// TwinCAT 3 PLC project PLC3
// ProgramVersion: 3.1.4022.3
// libraries:
//   Tc2_Standard, * (Beckhoff Automation GmbH)
//   Tc2_System, * (Beckhoff Automation GmbH)
//   Tc3_Module, * (Beckhoff Automation GmbH)
// project tree:
//   / CheckStatus.TcPOU, GlobalTextList.TcGTLO (not stored), PlcTask.TcTTO (not stored), Visualization Manager.TcVMO (not stored)
//   DUTs/ States.TcDUT
//   GVLs/ GVL_IO.TcGVL (not stored)
//   POUs/ MAIN.TcPOU, MoveArm.TcPOU

// ---- DUTs/States.TcDUT
{attribute 'qualified_only'}
{attribute 'strict'}
TYPE States :
(
	Init := 0,
	Idle,
	MoveToPickUp,
	PickUpDown,
	PickUpUp,
	Moving,
	DropDown,
	DropUp,
	PalletFull
);
END_TYPE

// ---- CheckStatus.TcPOU
FUNCTION_BLOCK CheckStatus
VAR_INPUT
	Position :INT;
	InputArray: ARRAY [1..25] OF BOOL;
END_VAR
VAR_OUTPUT
Occupied : BOOL;
END_VAR

Occupied := FALSE;
IF InputArray[Position] THEN
	Occupied := TRUE;
END_IF

END_FUNCTION_BLOCK

// ---- POUs/MAIN.TcPOU
PROGRAM MAIN
VAR
	Timer1 :TON;
	Timer2 : TON;
	Timer3 : TON;
	PulseTimer1 : TP;

	CurrentState  : States;
	
	ServoRTrigY : R_Trig ; 
	ServoRTrigX : R_Trig ; 
	
	//Eigen trigger booleans
	InitYReady : BOOL;
	InitXReady : BOOL;
	droppingDown : BOOL; //test
	
	TimerTest1 : TIME;
	TimerResult : TIME;
	
	Move_Arm : MoveArm;
	Check_Status : CheckStatus;
	
	PalletArray: ARRAY [1..25] OF BOOL := [25(FALSE)];

	Pos : INT;
END_VAR

PulseTimer1(IN:=GVL_IO.Start_button, PT:=T#150MS);
Timer1(IN:= GVL_IO.a_1_Vertical_Zaxis_downward, PT:= T#10MS);
Timer2(IN:=GVL_IO.a_1_Vertical_Zaxis_downward, PT:=T#10MS);
Timer3(IN:=droppingDown AND NOT GVL_IO.a_1_Vertical_Zaxis_downward, PT:=T#280MS);

CASE CurrentState OF
States.Init:
		//Aanzetten van servo's. Dit kan even duren GEEN HOMING
		GVL_IO.SVONX_SERVO_ON_tableX 	  := TRUE; 
		GVL_IO.SVONY_SERVO_ON_translY 	  := TRUE;
		
		GVL_IO.SETUPX_ORIGIN_tableX := PulseTimer1.Q;
		GVL_IO.SETUPY_ORIGIN_translY := PulseTimer1.Q;
		
		//// Koppelen van outputs Busy aan var's. Triggered op een falling edge.
		IF PulseTimer1.Q THEN
			ServoRTrigX ( clk := gvl_io.SETONX_ORIGIN_tableX ); 
	  		ServoRTrigY ( clk := gvl_io.SETONY_ORIGIN_translationY );
		END_IF
		
		// Bools setten aan de hand van triggers.
		IF ServoRTrigX.Q THEN
			InitXReady:= TRUE;
		END_IF
		
		IF ServoRTrigY.Q THEN
			InitYReady:= TRUE;
		END_IF
		
		// Init voltooid ga naar idle
		IF InitXReady AND InitYReady THEN
			Pos:= 1;
			CurrentState:= States.Idle;
		END_IF
		
States.Idle:
		IF NOT GVL_IO.Stop_button AND NOT GVL_IO.dp2_Cover_detection THEN
			//SEND MESSAGEE TODO
			CurrentState := States.Idle;
		END_IF
		
		IF NOT GVL_IO.Stop_button AND GVL_IO.dp1_Can_detection AND GVL_IO.dp2_Cover_detection THEN
			CurrentState := States.MoveToPickUp;
		END_IF
		
States.MoveToPickUp:
		Check_Status(Position:= POS, InputArray:= PalletArray);
		IF Check_Status.Occupied THEN
			CurrentState := States.ManualCheck;
			ELSE
				Move_Arm(Position:= 30);
				IF Move_Arm.OnNewLocation THEN
				CurrentState := States.PickUpDown;
				END_IF
		END_IF
		
States.PickUpDown:
		IF GVL_IO.a_0_Vertical_Zaxis_upward THEN
			GVL_IO.Aplus_Vert_axis_downwards := TRUE;
		END_IF
		
		IF GVL_IO.a_1_Vertical_Zaxis_downward THEN
			GVL_IO.Vplus_Vacuum_start := TRUE;
			
			IF Timer1.Q THEN
			CurrentState := States.PickUpUp;
			END_IF
		END_IF

States.PickUpUp:
		GVL_IO.Aplus_Vert_axis_downwards := FALSE;
		
		IF GVL_IO.a_0_Vertical_Zaxis_upward THEN
			CurrentState := States.Moving;
		END_IF
		
States.Moving:
		IF GVL_IO.a_0_Vertical_Zaxis_upward THEN
		
		Move_Arm(Position:= Pos);
		IF Move_Arm.OnNewLocation THEN
			PalletArray[Pos] := TRUE; // TEMP Cihan
			CurrentState := States.DropDown;
		END_IF
		END_IF
		
States.DropDown:
		IF GVL_IO.a_0_Vertical_Zaxis_upward THEN
			GVL_IO.Aplus_Vert_axis_downwards := TRUE;
			droppingDown := TRUE;
			TimerTest1 := TIME();
		END_IF
		
		
		IF 	GVL_IO.a_1_Vertical_Zaxis_downward THEN
			GVL_IO.Vplus_Vacuum_start := FALSE;
			IF Timer2.Q THEN
				TimerResult := TIME() - TimerTest1;
				droppingDown := FALSE;
				CurrentState := States.DropUp;
			END_IF
			
		ELSE IF Timer3.Q  THEN
		GVL_io.Aplus_Vert_axis_downwards := FALSE;
		droppingDown := FALSE;
		CurrentState := States.ManualCheck;
		END_IF
		END_IF

States.DropUp:
		IF GVL_IO.a_1_Vertical_Zaxis_downward THEN
			GVL_IO.Aplus_Vert_axis_downwards := FALSE;
		END_IF
		
		IF GVL_IO.a_0_Vertical_Zaxis_upward THEN
			CurrentState := States.Idle;
		END_IF
		
States.ManualCheck:
		GVL_IO.BR_Alarm_light := TRUE;
		GVL_io.Vplus_Vacuum_start := FALSE;
		IF GVL_IO.Reset_button THEN
			GVL_IO.BR_Alarm_light := FALSE;
			Currentstate := States.Idle;
		END_IF
END_CASE

END_PROGRAM

// ---- POUs/MoveArm.TcPOU
FUNCTION_BLOCK MoveArm
VAR_INPUT
Position: INT;
END_VAR
VAR_OUTPUT
	OnNewLocation:BOOL;
END_VAR
VAR
	X: INT;
	Y: INT;
	StartTimer:BOOL;
	
	
	PulseTimer2: TP;
	BusyFtrigX : F_Trig;
	BusyFtrigY : F_Trig;
	ReadyX : BOOL;
	ReadyY : BOOL;
	Busy: BOOL;
END_VAR

OnNewLocation := FALSE;

IF( Position < 1 OR Position > 30)  
	THEN RETURN; 
END_IF

// Calculate X & Y position on Palletiser
// 
X := (Position - 1) MOD 5;

// Position-1 / 5 with ROUND to floor 
Y := ((Position -1) / 5) - ((Position -1) / 5) MOD 1;

// set position 
GVL_IO.INX0_from_Input0_tableX:= X.0;
GVL_IO.INX1_from_Input1_tableX:= X.1;
GVL_IO.INX2_from_Input2_tableX:= X.2;
GVL_IO.INY0_from_Input0_translY:= Y.0;
GVL_IO.INY1_from_Input1_translY:= Y.1;
GVL_IO.INY2_from_Input2_translY:= Y.2;



PulseTimer2(IN:=StartTimer, PT:=T#150MS);

GVL_IO.DRIVEX_MOVE_tableX := PulseTimer2.Q;
GVL_IO.DRIVEY_MOVE_translY := PulseTimer2.Q;
StartTimer:= TRUE;
		
BusyFtrigX ( clk := gvl_io.BUSYX_BUSY_tableX ); 
BusyFtrigY ( clk := gvl_io.BUSYY_BUSY_traslationY );
		
IF BusyFtrigX.Q THEN
	ReadyX:= TRUE;
END_IF
		
IF BusyFtrigY.Q THEN
	ReadyY:= TRUE;
END_IF
		
IF ReadyY AND ReadyX THEN
	GVL_IO.DRIVEX_MOVE_tableX := FALSE;
	GVL_IO.DRIVEY_MOVE_translY := FALSE;
	ReadyX:= FALSE;
	ReadyY:= FALSE;
	StartTimer:= FALSE;
	OnNewLocation := TRUE;
END_IF

END_FUNCTION_BLOCK
